// TIA Portal V17 export
// export: Created 2024-08-09T12:53:23.1754197Z, ExportSetting WithDefaults, DisplayName Totally Integrated Automation Portal, DisplayVersion V17 Update 7, DisplayName TIA Portal Openness, DisplayVersion V17 Update 7, DisplayName TIA Portal Version Control Interface, DisplayVersion V17, DisplayName STEP 7 Professional, DisplayVersion V17 Update 7, DisplayName STEP 7 Safety, DisplayVersion V17 Update 6, DisplayName WinCC Professional, DisplayVersion V17 Update 7
TYPE "S_Commande"
// stored: IsFailsafeCompliant false
   STRUCT
      _CdMatOrg { ExternalAccessible := 'False'; ExternalVisible := 'False'; ExternalWritable := 'False'} : String["T_CD_MAT"];   // code mp Equivalente
      _LbMatOrg { ExternalAccessible := 'False'; ExternalVisible := 'False'; ExternalWritable := 'False'} : String["T_LB_MAT"];   // libelle mp Equivalente
      _CdMatComm { ExternalAccessible := 'False'; ExternalVisible := 'False'; ExternalWritable := 'False'} : String["T_CD_MAT"];   // code mp commandee
      _LbMatComm { ExternalAccessible := 'False'; ExternalVisible := 'False'; ExternalWritable := 'False'} : String["T_LB_MAT"];   // libelle mp commandee
      _Cel : String["T_CD_CEL"];   // code cellule
      _NoCommande { ExternalAccessible := 'False'; ExternalVisible := 'False'; ExternalWritable := 'False'} : String;
      _CdClient { ExternalAccessible := 'False'; ExternalVisible := 'False'; ExternalWritable := 'False'} : String;
      _NomClient { ExternalAccessible := 'False'; ExternalVisible := 'False'; ExternalWritable := 'False'} : String;
      _Ville { ExternalAccessible := 'False'; ExternalVisible := 'False'; ExternalWritable := 'False'} : String;
      _CdPost { ExternalAccessible := 'False'; ExternalVisible := 'False'; ExternalWritable := 'False'} : String;
      _Case { ExternalAccessible := 'False'; ExternalVisible := 'False'; ExternalWritable := 'False'} : String;
      _CdDepot { ExternalAccessible := 'False'; ExternalVisible := 'False'; ExternalWritable := 'False'} : String;   // Code Depot de la commande
      _Ni { ExternalAccessible := 'False'; ExternalVisible := 'False'; ExternalWritable := 'False'} : String;
      _NoLot { ExternalAccessible := 'False'; ExternalVisible := 'False'; ExternalWritable := 'False'} : String["T_Num_Lot"];   // Numero de lot
      _QteTotComm { ExternalAccessible := 'False'; ExternalVisible := 'False'; ExternalWritable := 'False'} : Real;
      _QteDejaCharg { ExternalAccessible := 'False'; ExternalVisible := 'False'; ExternalWritable := 'False'} : Real;
      _ChuteCel : Real;   // colonne de chute
      _DebitCel { ExternalAccessible := 'False'; ExternalVisible := 'False'; ExternalWritable := 'False'} : Real;   // Debit cellule
      _Densite { ExternalAccessible := 'False'; ExternalVisible := 'False'; ExternalWritable := 'False'} : Real;   // densite produit
      _VitGV : USInt;   // Vitesse variateur en GV
      _VitPV : USInt;   // Vitesse variateur en PV
      _SeuilPV : Real;   // poids pour passage en PV
      _NoLigne { ExternalAccessible := 'False'; ExternalVisible := 'False'; ExternalWritable := 'False'} : USInt;
      _IdComLig { ExternalAccessible := 'False'; ExternalVisible := 'False'; ExternalWritable := 'False'} : ULInt;
      _NmOrdre { ExternalAccessible := 'False'; ExternalVisible := 'False'; ExternalWritable := 'False'} : USInt;
      _NbCompo { ExternalAccessible := 'False'; ExternalVisible := 'False'; ExternalWritable := 'False'} : USInt;
      _AutrePont { ExternalAccessible := 'False'; ExternalVisible := 'False'; ExternalWritable := 'False'} : Bool;
   END_STRUCT;
END_TYPE
